// TIA Portal V20 export
FUNCTION "CallEnEffMonitor" : Void   // FC32, LAD
TITLE = CallEnergyEfficencyMonitor
AUTHOR : SICAR
FAMILY : Energy_EEM
VERSION : 1.0
// The S7 Energy Efficiency-Monitor (or S7 EE-Monitor) allows you to record the energy consumption of your machine in a SIMATIC controller, and to analyze the results on the basis of the energy and media requirements.
// stored: IsIECCheckEnabled true, SetENOAutomatically true
   VAR_TEMP
      tempMeasPointIndex : USInt;   // HMI index
      tempCycleCounterAvgCalc : DInt;   // Calculation to TOD
      tempPlantInProduction : Bool;   // Plant in production
      tempReturnValue : Int;   // Temporärer Wert zur Speicherung der EnPi-Resetzeit
   END_VAR
   // Ret_Val : Ret_Val
   VAR_TEMP   // added for the SCL form of the ladder/FBD networks
      _w1 : Bool;
      _w2 : Bool;
      _w3 : Bool;
      _w4 : Bool;
   END_VAR
BEGIN

REGION Network 1: BLOCK INFO HEADER
   // SIEMENS AG / (c)Copyright 2023
   // ------------------------------------------------------------------------------
   // Title:            CallEnEffMonitor (FC32)
   // Comment/Function: Call of Demo EnergyMeter and Energy Efficient M for EEMM demonstration
   // Library/Family:   Energy
   // Author:           SICAR
   // Tested with:      ---
   // Engineering:      TIA Portal V19
   // Restrictions:     -
   // Requirements:     ---
   // ------------------------------------------------------------------------------
   // Change log table:
   // Version  | Date       | Expert in charge       | Changes applied
   // ---------|------------|------------------------|------------------------------
   // 05.00.00 | 01.09.2023 | SICAR
   //                         First released version
END_REGION

REGION Network 2: DESCRIPTION
   // The Energy Efficiency Monitor “EEM” integrated in SICAR is based on the application example in entry ID: 109753230 V1.0 dated 02/2018 of the Siemens Industry Online Support, see: 
   // 
   // https://support.industry.siemens.com/cs/document/109753230/-s7-energy-efficiency-monitor-for-machines?dti=0&lc=en-WW 
   // 
   // **License**  
   // The software package has to be licensed. The necessary license key has to be entered in the data block for energy data “EEmData”, in the array item “licenseKey”. 
   //  
   // {.pageWidth}
   // ![Image](EemEnPiCalc/en/image1.PNG)
   // 
   // The S7 Energy Efficiency-Monitor (or S7 EE-Monitor) allows you to record the energy consumption of your machine in a SIMATIC controller, and to analyze the results on the basis of the energy and media requirements.  
   // https://support.industry.siemens.com/cs/document/109753230/s7-energieeffizienz-monitor-für-maschinen?dti=0&lc=de-WW 
   // 
   // **PLC Data types**  
   //  LSicar_typeEeMenPiCalc 
   //  LSicar_typeEeMenPiEstate 
   //  LSicar_typeEeMenPiLimit 
   //  typeEnMeterOutputData 
   //  typeMeasDataProfileE3 
   //  
   // **WinCC Faceplates**  
   // 
   // ![Image](EemEnPiCalc/en/image3.PNG)
   // 
   // **WinCC Screen**  
   //  
   // ![Image](EemEnPiCalc/en/image4.PNG)
   //  
   // # Devices & networks 
   // 
   // An additional AI Energy Meter has been added and configured in the SICAR project. The user data has been  
   // configured as module version “EE@Industry measured data profile e3”.  
   // 
   // Select the module version according to your requirements. The data assignment in the FC blocks has to be adjusted according to the selected module version. 
   // 
   // ![Image](EemEnPiCalc/en/image5.PNG)
   //  
   //  
   // 
   //  #### PLC Programm blocks 
   // 
   // ##### CallEnSeem  
   // The block is called in OB “CYCLIC_INTERRUPT_100MS_OB” (100ms cycle). The block contains the following instructions which can be found in “Instructions > Optional packages > Energy Suite extensions”.
   // 
   // **EnS_EEm_Calc:**  
   // The instruction calculates operating state-related energy data of machines and plants for uniform efficiency evaluation, in accordance with the VDMA 34179 measuring directive. 
   // 
   // ---
   // Note
   // :     The instruction calculates the energy efficiency value of the respective state for up to 8 operating states, and the global energy efficiency value. 
   // :     The maximum number of configurable measuring points is 10. Refer to the documentation of the entry ID. 
   // 
   // ---
   // 
   // **EnS_EEm_Report:**  
   // The instruction writes the data for the efficiency report to the data log on the SIMATIC memory card, in accordance with the VDMA 34179 measuring directive. The data log is a CSV file. 
   // 
   // ##### CallEnEffMonitor
   // ---
   // Note
   // :     The assignment of the readings as well as the formation of additional signals can be represented only exemplarily here. It has to be adapted to the actual plant conditions! 
   // 
   // ---
   // 
   // * Networks 1 & 2: The readings of the two AI-Energy-Meters are entered in the DB “EeMonitor”, in an array [0..9] in accordance with the measurement data profile “typeMeasDataProfileE3”. 
   // * Network 3: According to the selection of a measuring point on the HMI, data of the respective measuring point is routed to the HMI data area. The selection is done with a Pull-Down menu and a symbolic I/O field. 
   // * Network 4: Several tags in the EnS…data types are not marked as accessible / visible. In order to display these tags on the HMI all the same, they are routed to DB “EeMonitor” in structure “typeEnMeterWorkHmi”. There the tags are marked as accessible / visible.  
   // * Network 5: A collective signal is generated, according to the exemplary calls for OP area 1. This is only an example! The collective signal shows that the plant is producing parts, by a disjunction (OR) of all outputs. If an output is controlled, the plant is moving and producing parts. This collective signal is used later on to generate the energetic states “eState”. A delay of 3 seconds has been configured so that a short break in controlling the outputs will not change the energetic state. *
   // * Network 6: The signals for the energetic states are generated here. 
   // * Network 7: Simulation On/Off: A part counter is simulated here. Note: the simulation can be switched on and off with a button in the screen. 
   // * Network 8: Simulation On/Off. Energy counters for both AI-Energy-Meters are simulated here. Note: the simulation can be switched on and off with a button in the screen. 
   // * Network 9: Call of blocks “EemDemoSimulation” and “EemDemoResetValEMeter”. 
   // * Network 10: Call of block “EemEnPiCalc” and data routing according to the selection of a measuring point on the HMI. 
   // * Network 11: Error evaluation of block “EemEnPiCalc” to generate ProDiag messages. 
   // * Network 12: Error evaluation of block “EnS_EEm_Report” to generate ProDiag messages.  
   // 
   // ##### EemDemoResetValEMeter  
   // 
   // The block resets certain measurement values by controlling the respective outputs in the I/O area of the AI-Energy-Meter. 
   // 
   // ##### EemDemoSimulation  
   // 
   // This block simulates higher or lower energy values, according to the energetic states “eState”. 
   // 
   // ##### EemEnPiCalc
   // This block calculates the ENPI (Energy value Pro Item). It substitutes the script “EEm_EnPI_Efficiency” of the entry ID. 
   // 
   // ---
   // Note
   // :     All block parameters are provided with “pre-defined actual parameters”.
   // 
   // ---
   // 
   // **Operation mode Automatic / Manual**  
   // 
   // The blocks are independent of operation modes. Therefor they are not assigned to any operation mode area. 
   // 
   // **PLC Alarm text list**  
   // 
   // The following PLC alarm text lists have been created: 
   // 
   // * **EEMonitor_Calc_Warn_PD** ProDiag alarm text list for alarms by instruction “EnS_EEm_Calc”.   
   // * **EEMonitor_Report_Warn_PD** ProDiag alarm text list for alarms by instruction “EnS_EEm_Report”.   
   // Both PLC alarm text lists have been entered in the PLC alarm text list “GLOBAL_GENERAL_AlarmTextList”. 
   // 
   // ---
   // Note
   // :     The alarm texts are provided in two languages (German, English). Please consider the multilingual nature of the entries. 
   // 
   // ---
   // 
   // #### PLC Data types 
   // 
   // PLC data types used for PLC program block or HMI faceplate:  
   // ![Image](_Icon/reference.PNG)  See ..\Library Types\LSicar_typeEeMenPiCalc.pdf  
   // 
   // #### WinCC Objects 
   // 
   // **WinCC HMI-tags**  
   // 
   // The HMI tags are stored in the tag table “AI_EnergyMeter_EEM” in the SICAR project.  
   // 
   // **WinCC Text and graphics lists**  
   // 
   // The text list “EE-MONITOR_MEASUREPOINT” contains the texts necessary for the pull-down menu / symbolic I/O field in the screen. Please take into account the multilingual nature of the entries.  
   // 
   // **WinCC Faceplates**  
   // 
   // The faceplates are stored in the project library, in folder “types”. They have been created using several WinCC objects; they are animated depending on the state. 
   // 
   // * EEM_EnPI_EnergyPerItem:	display of ENPI (ENergy Per Item) 
   // * EEM_ViewBar_Diff-AVG-REF:	bar display to compare reference value and average value 
   // * EEM_ViewBar_EState-Total:	bar display of energy status (not used at this time) 
   // * EEM_ViewBarCurve_EState:	Total: bar display and curve display of the energy values  
   // 
   // **WinCC-screen** 
   // 
   // 1. HMI Screens:	EE-MONITOR_ENERGY: display of the energy values 
   // 2. HMI Popup-screens 
   // 	* EEM_LEGEND_Popup: 		Legend 
   // 	* EEM_INFO-MACHINE_Popup: 	Machine information 
   // 	* EEM_STARTMEASURE_Popup: 	Popup to start the normal measurement or the reference measurement  
   // 	* EEM_UIPE_Popup: 		display of voltage, current, power, and energy 
   // 	* MORE_EEM_Popup: 		Popup with additional buttons 
   // 	* MORE_AddOn_Popup: 		supplemented  with button “EE-Monitor” 
   // 
   //  
   // 
   // {.pageWidth}
   // ![Image](EemEnPiCalc/en/image6.PNG)
   //  
   //  
   // 
   // #### Additional information
   // 
   // #### Update info
   // 
   // #### Further documentations
END_REGION

REGION Network 3: select measurement values
   // can be from EnergyMeter driver or directly from any hardware (in this example EnergyMeter module and PAC)
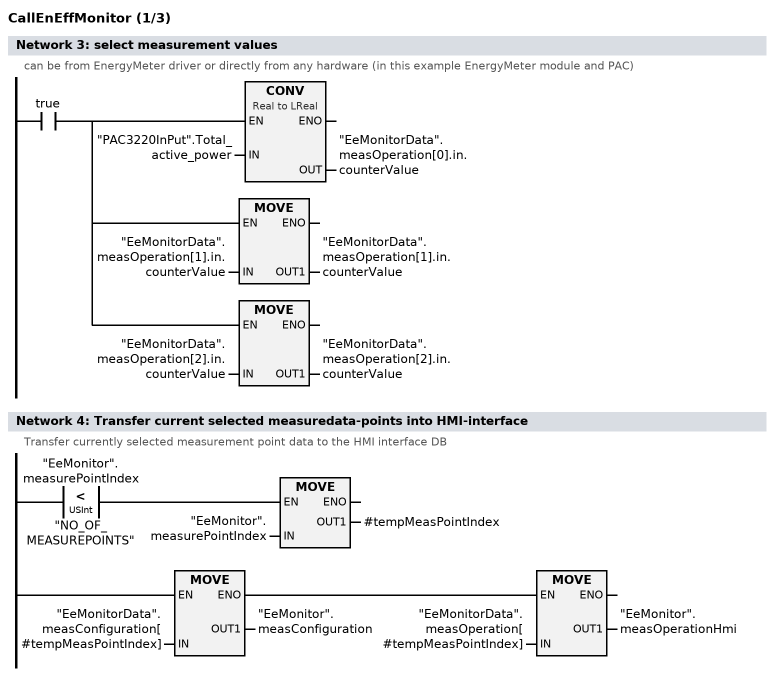
   RUNG wire#powerrail
      Contact( true )
      wire#w1
      { S7_Templates := "[SrcType := Real, DestType := LReal]" } Convert(in := "PAC3220InPut".Total_active_power, out => "EeMonitorData".measOperation[0].in.counterValue)
   END_RUNG
   RUNG wire#w1
      Move(in := "EeMonitorData".measOperation[1].in.counterValue, out1 => "EeMonitorData".measOperation[1].in.counterValue)
   END_RUNG
   RUNG wire#w1
      Move(in := "EeMonitorData".measOperation[2].in.counterValue, out1 => "EeMonitorData".measOperation[2].in.counterValue)
   END_RUNG
   // the same network as SCL:
   IF true THEN
       "EeMonitorData".measOperation[0].in.counterValue := REAL_TO_LREAL("PAC3220InPut".Total_active_power);
       "EeMonitorData".measOperation[1].in.counterValue := "EeMonitorData".measOperation[1].in.counterValue;
       "EeMonitorData".measOperation[2].in.counterValue := "EeMonitorData".measOperation[2].in.counterValue;
   END_IF;
END_REGION

REGION Network 4: Transfer current selected measuredata-points into HMI-interface
   // Transfer currently selected measurement point data to the HMI interface DB
   RUNG wire#powerrail
      { S7_Templates := "SrcType := USInt" } LT_Contact(in1 := "EeMonitor".measurePointIndex, in2 := "NO_OF_MEASUREPOINTS")
      Move(in := "EeMonitor".measurePointIndex, out1 => #tempMeasPointIndex)
   END_RUNG
   RUNG wire#powerrail
      Move(in := "EeMonitorData".measConfiguration[#tempMeasPointIndex], out1 => "EeMonitor".measConfiguration)
      Move(in := "EeMonitorData".measOperation[#tempMeasPointIndex], out1 => "EeMonitor".measOperationHmi)
   END_RUNG
   // the same network as SCL:
   IF "EeMonitor".measurePointIndex < "NO_OF_MEASUREPOINTS" THEN
       #tempMeasPointIndex := "EeMonitor".measurePointIndex;
   END_IF;
   "EeMonitor".measConfiguration := "EeMonitorData".measConfiguration[#tempMeasPointIndex];
   "EeMonitor".measOperationHmi := "EeMonitorData".measOperation[#tempMeasPointIndex];
END_REGION

REGION Network 5: WORKaround: Transfer data from EeMonitroData to EeMonitor.work
   // Convertion of Time to DTL and adding time zone with date and time taken from EnS_EEm_Calc for representing the actual date and time in the current country.
   // Data is copied from EeMonitorData to EeMonitor.work
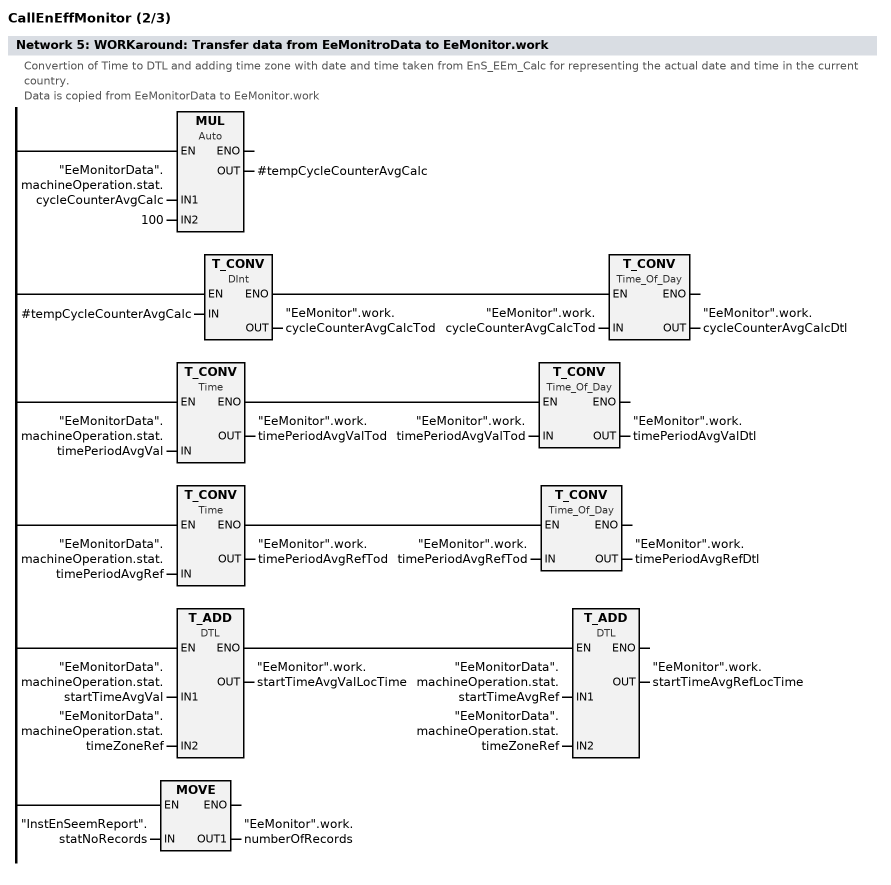
   RUNG wire#powerrail
      Mul(in1 := "EeMonitorData".machineOperation.stat.cycleCounterAvgCalc, in2 := 100, out => #tempCycleCounterAvgCalc)
   END_RUNG
   RUNG wire#powerrail
      { S7_Templates := "[src_type := DInt, dest_type := Time_Of_Day]" } T_CONV(IN := #tempCycleCounterAvgCalc, OUT => "EeMonitor".work.cycleCounterAvgCalcTod)
      { S7_Templates := "[src_type := Time_Of_Day, dest_type := DTL]" } T_CONV(IN := "EeMonitor".work.cycleCounterAvgCalcTod, OUT => "EeMonitor".work.cycleCounterAvgCalcDtl)
   END_RUNG
   RUNG wire#powerrail
      { S7_Templates := "[src_type := Time, dest_type := Time_Of_Day]" } T_CONV(IN := "EeMonitorData".machineOperation.stat.timePeriodAvgVal, OUT => "EeMonitor".work.timePeriodAvgValTod)
      { S7_Templates := "[src_type := Time_Of_Day, dest_type := DTL]" } T_CONV(IN := "EeMonitor".work.timePeriodAvgValTod, OUT => "EeMonitor".work.timePeriodAvgValDtl)
   END_RUNG
   RUNG wire#powerrail
      { S7_Templates := "[src_type := Time, dest_type := Time_Of_Day]" } T_CONV(IN := "EeMonitorData".machineOperation.stat.timePeriodAvgRef, OUT => "EeMonitor".work.timePeriodAvgRefTod)
      { S7_Templates := "[src_type := Time_Of_Day, dest_type := DTL]" } T_CONV(IN := "EeMonitor".work.timePeriodAvgRefTod, OUT => "EeMonitor".work.timePeriodAvgRefDtl)
   END_RUNG
   RUNG wire#powerrail
      { S7_Templates := "[date_type := DTL, time_type := Time]" } T_ADD(IN1 := "EeMonitorData".machineOperation.stat.startTimeAvgVal, IN2 := "EeMonitorData".machineOperation.stat.timeZoneRef, OUT => "EeMonitor".work.startTimeAvgValLocTime)
      { S7_Templates := "[date_type := DTL, time_type := Time]" } T_ADD(IN1 := "EeMonitorData".machineOperation.stat.startTimeAvgRef, IN2 := "EeMonitorData".machineOperation.stat.timeZoneRef, OUT => "EeMonitor".work.startTimeAvgRefLocTime)
   END_RUNG
   RUNG wire#powerrail
      Move(in := "InstEnSeemReport".statNoRecords, out1 => "EeMonitor".work.numberOfRecords)
   END_RUNG
   // the same network as SCL:
   #tempCycleCounterAvgCalc := "EeMonitorData".machineOperation.stat.cycleCounterAvgCalc * 100;
   T_CONV(IN := #tempCycleCounterAvgCalc, OUT => "EeMonitor".work.cycleCounterAvgCalcTod, ENO => #_w1);
   IF #_w1 THEN
       T_CONV(IN := "EeMonitor".work.cycleCounterAvgCalcTod, OUT => "EeMonitor".work.cycleCounterAvgCalcDtl);
   END_IF;
   T_CONV(IN := "EeMonitorData".machineOperation.stat.timePeriodAvgVal,
          OUT => "EeMonitor".work.timePeriodAvgValTod,
          ENO => #_w2);
   IF #_w2 THEN
       T_CONV(IN := "EeMonitor".work.timePeriodAvgValTod, OUT => "EeMonitor".work.timePeriodAvgValDtl);
   END_IF;
   T_CONV(IN := "EeMonitorData".machineOperation.stat.timePeriodAvgRef,
          OUT => "EeMonitor".work.timePeriodAvgRefTod,
          ENO => #_w3);
   IF #_w3 THEN
       T_CONV(IN := "EeMonitor".work.timePeriodAvgRefTod, OUT => "EeMonitor".work.timePeriodAvgRefDtl);
   END_IF;
   T_ADD(IN1 := "EeMonitorData".machineOperation.stat.startTimeAvgVal,
         IN2 := "EeMonitorData".machineOperation.stat.timeZoneRef,
         OUT => "EeMonitor".work.startTimeAvgValLocTime,
         ENO => #_w4);
   IF #_w4 THEN
       T_ADD(IN1 := "EeMonitorData".machineOperation.stat.startTimeAvgRef,
             IN2 := "EeMonitorData".machineOperation.stat.timeZoneRef,
             OUT => "EeMonitor".work.startTimeAvgRefLocTime);
   END_IF;
   "EeMonitor".work.numberOfRecords := "InstEnSeemReport".statNoRecords;
END_REGION

REGION Network 6: Operation modes to "eState"
   // Sets Estate number accoriding to the selected state
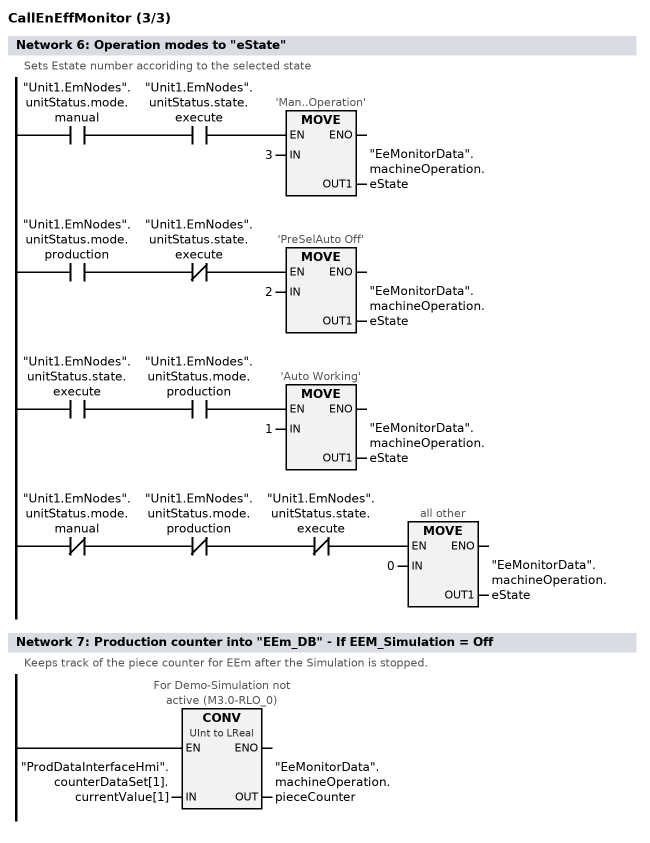
   RUNG wire#powerrail
      Contact( "Unit1.EmNodes".unitStatus.mode.manual )
      Contact( "Unit1.EmNodes".unitStatus.state.execute )
      Move(in := 3, out1 => "EeMonitorData".machineOperation.eState)   // 'Man..Operation'
   END_RUNG
   RUNG wire#powerrail
      Contact( "Unit1.EmNodes".unitStatus.mode.production )
      I_Contact( "Unit1.EmNodes".unitStatus.state.execute )
      Move(in := 2, out1 => "EeMonitorData".machineOperation.eState)   // 'PreSelAuto Off'
   END_RUNG
   RUNG wire#powerrail
      Contact( "Unit1.EmNodes".unitStatus.state.execute )
      Contact( "Unit1.EmNodes".unitStatus.mode.production )
      Move(in := 1, out1 => "EeMonitorData".machineOperation.eState)   // 'Auto Working'
   END_RUNG
   RUNG wire#powerrail
      I_Contact( "Unit1.EmNodes".unitStatus.mode.manual )
      I_Contact( "Unit1.EmNodes".unitStatus.mode.production )
      I_Contact( "Unit1.EmNodes".unitStatus.state.execute )
      Move(in := 0, out1 => "EeMonitorData".machineOperation.eState)   // all other
   END_RUNG
   // the same network as SCL:
   IF "Unit1.EmNodes".unitStatus.mode.manual AND "Unit1.EmNodes".unitStatus.state.execute THEN
       "EeMonitorData".machineOperation.eState := 3;   // 'Man..Operation'
   END_IF;
   IF "Unit1.EmNodes".unitStatus.mode.production AND NOT "Unit1.EmNodes".unitStatus.state.execute THEN
       "EeMonitorData".machineOperation.eState := 2;   // 'PreSelAuto Off'
   END_IF;
   IF "Unit1.EmNodes".unitStatus.state.execute AND "Unit1.EmNodes".unitStatus.mode.production THEN
       "EeMonitorData".machineOperation.eState := 1;   // 'Auto Working'
   END_IF;
   IF NOT "Unit1.EmNodes".unitStatus.mode.manual AND NOT "Unit1.EmNodes".unitStatus.mode.production AND NOT "Unit1.EmNodes".unitStatus.state.execute THEN
       "EeMonitorData".machineOperation.eState := 0;   // all other
   END_IF;
END_REGION

REGION Network 7: Production counter into "EEm_DB" - If EEM_Simulation = Off
   // Keeps track of the piece counter for EEm after the Simulation is stopped.
   RUNG wire#powerrail
      { S7_Templates := "[SrcType := UInt, DestType := LReal]" } Convert(in := "ProdDataInterfaceHmi".counterDataSet[1].currentValue[1], out => "EeMonitorData".machineOperation.pieceCounter)   // For Demo-Simulation not active (M3.0-RLO_0)
   END_RUNG
   // the same network as SCL:
   "EeMonitorData".machineOperation.pieceCounter := UINT_TO_LREAL("ProdDataInterfaceHmi".counterDataSet[1].currentValue[1]);   // For Demo-Simulation not active (M3.0-RLO_0)
END_REGION

REGION Network 8 (SCL): Reset EnPI values
   // Reads the current time and store it to provide the user the information about the last EnPi reset
   // Check for the trigger to reset/recalculate the EnPI values
   IF ("EeMonitorData".internalData.enpiResetTrigger = TRUE) THEN

       // Read the current time and store it to provide the user the information
       // about the last reset
       #tempReturnValue := RD_LOC_T("EeMonitorData".internalData.enpiResetTime);

       // Reset the trigger
       "EeMonitorData".internalData.enpiResetTrigger := FALSE;
   ELSE
       ; // No trigger
   END_IF;
END_REGION
END_FUNCTION
